(* PLC project PLC_Project, Beckhoff Automation GmbH TwinCAT PLC Control 3.5.13.21 *)
(* stored: creationDateTime 2023-07-15T20:01:09.8640191, modificationDateTime 2023-07-15T20:01:09.8669938 *)

FUNCTION_BLOCK FB_PULSO
VAR_INPUT
	Referencia_a_variable_a_Pulsar: REFERENCE TO BOOL;
	Temps_pols : TIME;	
END_VAR
VAR_OUTPUT

END_VAR
VAR
	TP1: TP;
	Activar_TP1 : BOOL;
	Temps : TIME;
	Temps_actual_pols : TIME;
	Variable_pulsdada : BOOL;
END_VAR

               



     TP1(IN:= Referencia_a_variable_a_Pulsar , PT:=  Temps_pols, Q=> Variable_pulsdada   , ET=> Temps_actual_pols  );
	IF TP1.ET = TP1.PT THEN Referencia_a_variable_a_Pulsar := FALSE ;
		// <
	END_IF
	 
          
END_FUNCTION_BLOCK
